# EPICS autosave request: softglue/softGlueApp/Db/softGlue_FPGAContent_Encoder_settings.req
# up/dn counters and quadrature decoders
file UpDnCntr_settings.req P=$(P),H=$(H),N=1
file UpDnCntr_settings.req P=$(P),H=$(H),N=2
file QuadDec_settings.req P=$(P),H=$(H),N=1
file QuadDec_settings.req P=$(P),H=$(H),N=2

# descriptions
$(P)$(H)UpDnCntr-1_desc
$(P)$(H)UpDnCntr-2_desc
$(P)$(H)QuadDec-1_desc
$(P)$(H)QuadDec-2_desc
